	stParDutyCycle.fMinimum 		:= 0 		;
	stParDutyCycle.fMaximum			:= 50 		;
	stParDutyCycle.nNumber 			:= nLocationId + 2;
	stParDutyCycle.sDiscription  	:= CONCAT( STR1 := sName, STR2 := 'Percentage of period length in which an output is active');
	stParDutyCycle.sName			:= CONCAT( STR1 := sName, STR2 := 'Duty Cyle');
	stParDutyCycle.sType			:= 'MPar';
	stParDutyCycle.sUnit			:= '%';
	stParPeriodLength.fValue		:= 10;

	
	stParSwitchOverTime.fMinimum 	:= 0 		;
	stParSwitchOverTime.fMaximum	:= 500 		;
	stParSwitchOverTime.nNumber 	:= nLocationId + 3;
	stParSwitchOverTime.sDiscription:= CONCAT( STR1 := sName, STR2 := 'Idle time between output chanel switchover in miliseconds');
	stParSwitchOverTime.sName		:= CONCAT( STR1 := sName, STR2 := 'Switch Time');
	stParSwitchOverTime.sType		:= 'CPar';
	stParSwitchOverTime.sUnit		:= 'ms';

	stMaxTimeOn.fMinimum 	:= 0 		;
	stMaxTimeOn.fMaximum	:= 5000 	;
	stMaxTimeOn.nNumber 	:= nLocationId + 4;
	stMaxTimeOn.sDiscription:= CONCAT( STR1 := sName, STR2 := 'Maximum time a heater can be fully on without burning through');
	stMaxTimeOn.sName		:= CONCAT( STR1 := sName, STR2 := 'Max heating time');
	stMaxTimeOn.sType		:= 'MPar';
	stMaxTimeOn.sUnit		:= 'ms';
	
	
	// add parameters to handler 
	refFbParHandler.CmdAddParameter( refParameter := stParPeriodLength );
	refFbParHandler.CmdAddParameter( refParameter := stParDutyCycle );
	refFbParHandler.CmdAddParameter( refParameter := stParSwitchOverTime );
	
// ====== Set init status bit =======
	bInitOk := TRUE ;
END_METHOD

END_FUNCTION_BLOCK

// ---- Encoders/FunctionBlocks/FB_EncoderBase.TcPOU
{attribute 'reflection'}
FUNCTION_BLOCK PUBLIC FB_EncoderBase EXTENDS FB_DevBase
VAR_INPUT
END_VAR
VAR_OUTPUT
	{attribute 'analysis' := '-33'}
	nOutPosition		: LREAL	:= 0	; // Scaled position output
	{attribute 'analysis' := '-33'}
	nOutRaw				: UDINT := 0	; // Raw output value
	{attribute 'analysis' := '-33'}
	nVelocity			: LREAL	:= 0 	; // Velocity [units/sec]
END_VAR
VAR
	fPulsesPerUnit		: LREAL := 1	; // Scale factor for output [units/pulse]
	fOffset				: LREAL := 0	; // Offset for output
	bIcfInverted		: BOOL	:= FALSE; // Invert output position = standard false  
END_VAR

METHOD PUBLIC FastTask : BOOL
VAR_INPUT
END_VAR
END_METHOD

METHOD PUBLIC Init : BOOL
VAR_INPUT
	// Message location data
	nId			: UDINT ; // Identification number of object
	nParentId	: UDINT ; // Id of higher level If aplicable (0 = no parent)
	// Configuration
	fPulsesPerUnit	: LREAL	; // Scale factor for output [units/pulse]
	fOffset			: LREAL	; // Offset for output
	bIcfInverted	: BOOL	; // Invert output position = standard false  
END_VAR


// ====== Calculate device id =====
	ExecIdentifyDevice(nId,nParentId, E_ComponentTypes.Encoder);

// ====== Set manual device type ======
	eDevType := E_Devices.Encoder ;	

	
// ===== Coppy values to function memory ======
	THIS^.fPulsesPerUnit	:= MAX(fPulsesPerUnit,0.01); // Minimum value of 1
	THIS^.fOffset			:= fOffset;
	THIS^.bIcfInverted		:= bIcfInverted;
	
	
bInitOk := TRUE ;
END_METHOD

END_FUNCTION_BLOCK

// ---- Axis/FunctionBlocks/Analog/FB_DevAnalogAxis.TcPOU
FUNCTION_BLOCK PUBLIC FB_DevAnalogAxis EXTENDS FB_DevBase
VAR_INPUT
	stManualCtrl 	: ST_ManualAnalogAxisCtrl ; // Manual control
END_VAR
VAR_OUTPUT
	bDriveOk		: BOOL ; // Drive is ok
	bMovingCW		: BOOL ; // Move CW output is active
	bMovingCCW		: BOOL ; // Move CCW output is active
	fActVelocity	: LREAL; // Command velocity of motor
END_VAR
VAR // internal functions 
	fbVelocity		: FB_DevAnalogOutputScaled 	;
	fbqRun			: FB_DevDigitalOutput		;
	fbqReset		: FB_DevDigitalOutput		;
	fbqReverse		: FB_DevDigitalOutput		;
	fbiEnabled		: Fb_DevDigitalInput		;
END_VAR
VAR // Internal commands
	fCmdVelocity	: LREAL;
	bCmdRunCW 		: BOOL ;
	bCmdRunCCW		: BOOL ;
	bCmdReset		: BOOL ;	 
	bInternalEnable : BOOL ;
END_VAR

SUPER^(refFbFault := refFbFault);

// ===== Check inputs =====
	fbiEnabled( bEmbeded	:= TRUE,
				refFbFault 	:= refFbFault);

IF bInitOk THEN 
	ExecSetOutputs() ;
	bDriveOk	:= fbiEnabled.bFcoInputActive ;
END_IF

METHOD PUBLIC CmdManual : BOOL
VAR_INPUT
END_VAR
bCmdManual := TRUE ;

// Execute Manual commands
	IF stManualCtrl.bCmdRunCW THEN 
		CmdRunCW(fCmdVelocity := stManualCtrl.fCmdVelocity);
	ELSIF stManualCtrl.bCmdRunCCW THEN 
		CmdRunCCW(fCmdVelocity := stManualCtrl.fCmdVelocity);
	END_IF
END_METHOD

METHOD PUBLIC CmdReset : BOOL
VAR_INPUT
END_VAR
bErrorActive 	:= FALSE;

bCmdReset		:= TRUE ;

CmdReset		:= TRUE ;
END_METHOD

METHOD PUBLIC CmdRunCCW : BOOL
VAR_INPUT
	fCmdVelocity	: LREAL ; // Command velocity
END_VAR
bCmdRunCCW			:= TRUE ;
THIS^.fCmdVelocity 	:= fCmdVelocity ; 

CmdRunCCW 	:= bMovingCW ;
END_METHOD

METHOD PUBLIC CmdRunCW : BOOL
VAR_INPUT
	fCmdVelocity	: LREAL ; // Command velocity
END_VAR
bCmdRunCW := TRUE ;
THIS^.fCmdVelocity 	:= fCmdVelocity ;

CmdRunCW 	:= bMovingCW ;
END_METHOD

METHOD PUBLIC CmdSafeStop : BOOL
VAR_INPUT
END_VAR
bIsSafe := TRUE ;

bIsSafe := fbVelocity.CmdSafeStop() AND bIsSafe ;
bIsSafe := fbqRun.CmdSafeStop() 	AND bIsSafe ;
bIsSafe := fbqReverse.CmdSafeStop() AND bIsSafe ;
bIsSafe := fbqReset.CmdSafeStop() 	AND bIsSafe ;

CmdSafeStop := bIsSafe;
END_METHOD

METHOD PRIVATE ExecSetOutputs : BOOL
VAR_INPUT
END_VAR
// ====== Check safety and enable ======
IF bSafetyOk 
AND fbiEnabled.bFcoInputActive 
AND (bEnable OR bManual) THEN 
	bInternalEnable := TRUE;
ELSE
	fCmdVelocity 	:= 0;
	bCmdRunCW		:= FALSE;
	bCmdRunCCW		:= FALSE;
END_IF 

// ====== Set outputs =======
	fbVelocity	(	bEmbeded 	:= TRUE,
					bSafetyOk	:= bSafetyOk,
					bEnable		:= bInternalEnable,
					fCmdValue	:= fCmdVelocity, 
					refFbFault	:= refFbFault);
				
	fbqRun		(	bEmbeded 	:= TRUE,
					bSafetyOk	:= bSafetyOk,
					bEnable		:= bInternalEnable,
					bCmdOn		:= bCmdRunCW OR bCmdRunCCW,
					refFbFault	:= refFbFault);
				
	fbqReverse	(	bEmbeded 	:= TRUE,
					bSafetyOk	:= bSafetyOk,
					bEnable		:= bInternalEnable,
					bCmdOn		:= bCmdRunCCW,
					refFbFault	:= refFbFault);

	fbqReset	(	bEmbeded 	:= TRUE,
					bSafetyOk	:= bSafetyOk,
					bEnable		:= bInternalEnable,
					bCmdOn		:= bCmdReset,
					refFbFault	:= refFbFault);

// ===== reset input commands =====
	fCmdVelocity 	:= 0;
	bCmdRunCW		:= FALSE;
	bCmdRunCCW		:= FALSE;
	bCmdManual		:= FALSE;
	bCmdReset		:= FALSE;
	bInternalEnable := FALSE;
// ===== set feedback =====

bMovingCW		:= fbqRun.bOutputState AND NOT fbqReverse.bOutputState;
bMovingCCW		:= fbqRun.bOutputState AND fbqReverse.bOutputState;
fActVelocity	:= fbVelocity.fOutputValue ;
END_METHOD

METHOD Init : BOOL
VAR_INPUT
	// Message location data
	nId			: UDINT ; // Identification number of object
	nParentId	: UDINT ; // Id of higher level If aplicable (0 = no parent)

	// Motor settings
	fMaxVelocity : LREAL ; // Maximum motor velocity for scaling
END_VAR
// ====== initialize components =====
	bInitOk := TRUE ;

// ====== Calculate device id =====
	bInitOk :=	ExecIdentifyDevice(nId,nParentId, E_ComponentTypes.Axis) AND bInitOk;

// ====== Set manual device type ======
	eDevType := E_Devices.AnalogAxis ;	


bInitOk := 	fbVelocity.Init	( 	nId 			:= 0,
								nParentId		:= nLocationId,
								benableNegative	:= FALSE )
								AND bInitOk;
			fbVelocity.SetScaling	(fMaxValue 		:= fMaxVelocity);
								
bInitOk	:= 	fbqRun.Init		( 	nId				:= 1,
								nParentId		:= nLocationId)
								AND bInitOk;

bInitOk	:= 	fbqReset.Init	( 	nId				:= 2,
								nParentId		:= nLocationId)
								AND bInitOk;

bInitOk	:= 	fbqReverse.Init	( 	nId				:= 3,
								nParentId		:= nLocationId)
								AND bInitOk;

bInitOk	:= 	fbiEnabled.Init	( 	nId				:= 4,
								nParentId		:= nLocationId)
								AND bInitOk;

// ====== Set feedback =======
Init := bInitOk;
END_METHOD

END_FUNCTION_BLOCK

// ---- Outputs/AnalogOutputs/FB_DevAnalogOutputScaled.TcPOU
{attribute 'reflection'}
FUNCTION_BLOCK FB_DevAnalogOutputScaled EXTENDS FB_DevAnalogOutput
VAR_INPUT
END_VAR
VAR_OUTPUT
END_VAR
VAR
	fGainFactor 	: LREAL:= 32767	;
END_VAR

SUPER^(refFbFault := refFbFault);

METHOD INTERNAL ExecSetFeedback : BOOL
VAR_INPUT
END_VAR
// Set feedback 
fOutputValue := qnHwOut ;
END_METHOD

METHOD INTERNAL ExecSetOutput : BOOL
VAR_INPUT
END_VAR
// Set Output to physical device
IF bSafetyOk AND (bEnable OR bCmdManual) THEN 
	qnHwOut := LREAL_TO_INT(fCmdValue * fGainFactor) ;
	qnHwOut := LIMIT(nLimitMin, qnHwOut, nLimitMax) ; 
ELSE 
	qnHwOut		:= 0;
	fCmdValue 	:= 0 ; 
END_IF
END_METHOD

METHOD PUBLIC SetScaling : BOOL 
VAR_INPUT
	fMaxValue	: LREAL ; 		// Maximum input value after scaling, e.g. 100% (mandatory input)  
END_VAR
// calculate gain 
fGainFactor := nLimitMax / fMaxValue ;
END_METHOD

END_FUNCTION_BLOCK

// ---- Axis/FunctionBlocks/ServoHybrid/FB_DevBasicACAxis.TcPOU
{attribute 'reflection'}
FUNCTION_BLOCK PUBLIC FB_DevBasicACAxis EXTENDS FB_DevBase
VAR_INPUT
	// ===== General Function input =====
		fCmdAcc			: LREAL := 15000;
		fCmdDecc		: LREAL := 15000; 
	// Manual control reference
		stManualCtrl	: UDT_ManualAxisCtrl ;
END_VAR
VAR_OUTPUT
	bHomed			: BOOL 	:= FALSE; 
	bMoving		: BOOL ; // Axis is moving
	bInPosition : BOOL ; // Axis is in position 
END_VAR
VAR
		AxisRef	: AXIS_REF ; // reference to AC axis
	// ===== HW Config Bits =====
		bIcfCmdVelocityRpm	: BOOL ; // input speeds in Rpm
		bIcfEnableForward 	: BOOL ; // Enable forward motion
 		bIcfEnablereverse	: BOOL ; // Enable reverse motion
		bIcfAlwaysEnable	: BOOL ; // 1 = Axis always enabled, 0 = Axis disabled at Idle 
		bIcfSimulationMode	: BOOL := FALSE ; // Simulation mode is active [default set to False] 
	// ===== Internal motion values ======
		fHomePosition		: LREAL := 0 ; // set position at homing
	// ====== Axis Settings ======
		fMaxVelo		: LREAL := 0 ; // Axis Maximum velocity
		fMaxAcc			: LREAL := 0 ; // Axis Maximum cceleration
		fMaxDec			: LREAL := 0 ; // axis Maxium deceleration 
		
		fSafeVeloLimit	: LREAL	:= 200; // Safe velocity limit 
		tEnableDelay	: TIME 	:= T#150MS	;
		tDisableDelay	: TIME 	:= T#500MS  ;
		
	// ====== Axis enable =====	
		bCmdEnableAxis 		: BOOL 	:= FALSE; // Command to enable the axis (External)
		bInternalEnable		: BOOL 	:= FALSE; // internal enable command (turns off after set time, and on at new motion command
		bDelayedEnable		: BOOL 	:= false; // Delayed enable signal for motion commands
		TonMotionEnable		: TON 			; // Timer on for motion command enable
		TofIntAxisEnable	: TOF  			; // Timer off for internal axis enable 
	// ===== Safe commands =====
		bCmdSafeStop	: BOOL ;
	// Motion commands 
		fbMcPower 			: MC_Power		;		// FB for enable and override
		fbMcReset 			: MC_Reset		;		// FB to reset axis
		fbSoeReset			: FB_SoEReset	; 		// FB to reset axis hardware
		fbMcHome			: MC_Home		;		// Fb to home Axis
		fbMcStop 			: MC_Stop		;		// FB to stop axis
		fbMcHalt			: MC_Halt		;		// FB to halt axis
		fbMcJog				: MC_Jog		;		// FB to Jog axis
		fbMcMoveVelocity	: MC_MoveVelocity;		// FB to move with specified velocity until Next command is given
	(* PtoP Motion move commands are in arrays so multiple commands can be stacked *) 
		fbMCMoveRelative	: ARRAY [0..1] OF MC_MoveRelative	;		// FB to move relative
		fbMcMoveAbsolute	: ARRAY [0..1] OF MC_MoveAbsolute	;		// FB to move axis (velocity movement)
		
	// Parameters 
		stMParMaxAcc : Udt_Parameter := (fMaximum := 999999, fMinimum := 0, fValue := 0)	; // Parameter for maximum acceleration
		stMParMaxDec : Udt_Parameter := (fMaximum := 999999, fMinimum := 0, fValue := 0)	; // Parameter for maximum Deceleration
		stMparMaxVelo: Udt_Parameter := (fMaximum := 999999, fMinimum := 0, fValue := 0)	; // Parameter for maximum velocity
		
	// Device feedback
		nActVelocity AT%I* : INT ; // actual speed of the motor
		nActPosition AT%I* : UDINT ; // Actual position of the motor

	// ===== Function execute triggers =====
		bExec_Reset			: BOOL := FALSE; // Execute reset
		bExec_Halt			: BOOL := FALSE; // Execute hold
		bExec_Home			: BOOL := FALSE; // Execute Home
		bExec_JogPositive	: BOOL := FALSE; // Execute Jog in positive direction
		bExec_JogNegative	: BOOL := FALSE; // Execute Jog in negative direction
		bExec_MoveVelocity	: BOOL := FALSE; // Execute move velocity
		arExec_MoveRelative	: ARRAY [0..1] OF BOOL ; // Execute move relative
		arExec_MoveAbs		: ARRAY [0..1] OF BOOL ; // Execute move absolute reverse
		

END_VAR

// Call base function
SUPER^(refFbFault := refFbFault);

// ==== Check if axis is initiated =====
IF NOT bInitOk THEN 
	RETURN ; 
END_IF

// ===== Execute safe functions =====
	ExecSafeFunctions(); 

// ==== Execute organizational functions =====
	ExecEnable();

// ==== execute motion functions =====
	CallMotionFunctions();

METHOD PRIVATE CallMotionFunctions : BOOL
VAR_INPUT
END_VAR
// ===== Check if safe to move =====
	IF bCmdSafeStop OR NOT bDelayedEnable THEN 
		RETURN ;
	END_IF

// ===== Homing functions =====
	ExecHome		(); 

// ===== Motion standstil commands =====
	ExecHalt		();

// ===== Motion move functions
	ExecJog			(); 
	ExecMoveAbsolute();
	ExecMoveRelative();
	ExecMoveVelocity();
END_METHOD

METHOD PUBLIC CmdHalt : BOOL
VAR_INPUT
	fDeceleration 	: LREAL := 0 ; // command deceleration
	mcBuffermode	: MC_BufferMode ; // Buffermode defines how the previous command is executed.
END_VAR
// Set command to true 
bExec_Halt 		:= TRUE ;
bInternalEnable	:= TRUE ;

// coppy parameters
fbMcHalt.Deceleration	:= fDeceleration;
fbMcHalt.BufferMode		:= mcBuffermode	;

// Set feedback output 
CmdHalt := fbMchalt.Active ;
END_METHOD

METHOD PUBLIC CmdHome : BOOL // start axis homing procedure
VAR_INPUT
	fPosition 		: LREAL := 0 ; // Homing position
	mcBufferMode	: MC_BufferMode := MC_BufferMode.MC_Aborting		; // Buffermode
END_VAR
// set command to true 
bExec_Home 		:= TRUE	; 
bInternalEnable	:= TRUE ;

// coppy parameters
fbMcHome.Position 	:= fPosition 	;
fbMcHome.BufferMode	:= mcBufferMode ;

// Set feedback output
CmdHome := fbMcHome.Done ;
END_METHOD

METHOD PUBLIC CmdJog : BOOL // Jog axis with variable speed. jog stops as soon as the command is false
VAR_INPUT
	fVelocity		: LREAL 	; // jog velocity can be adjusted as long as the command is active
	fPos			: LREAL 	; // Jog position or step size (if aplicable)
	bJogNegative 	: BOOL 		:= FALSE ; // jog in negative direction
	eJogmode		: E_JogMode := E_JogMode.MC_JOGMODE_CONTINOUS ; // jogmode [default MC_JOGMODE_CONTINOUS] 
END_VAR
// Velocity conversion from RPM to deg/sec
	IF bIcfCmdVelocityRpm THEN 
		fVelocity := Rpm_To_DegS(fVelocity);
	END_IF

// Set command to true
	IF fbMcJog.Velocity = fVelocity THEN // If command velocity changes, then set exec to false for one cycle to trigger new velocity so the jog follows the set velocity
		bExec_JogPositive	:= NOT bJogNegative ;
		bExec_JogNegative 	:= bJogNegative ;
	END_IF
	bInternalEnable			:= TRUE ;

// coppy parameters
	fbMcJog.Velocity	:= fVelocity 	;
	fbmcjog.Mode		:= eJogmode		;
	fbMcJog.Position	:= fPos			;

// Set feedback output 
	CmdJog := fbMcJog.Active ;
END_METHOD

METHOD PUBLIC CmdManual : BOOL
VAR
	eJogmode		: E_JogMode := E_JogMode.MC_JOGMODE_CONTINOUS ; // jogging mode 
END_VAR
// Enable axis for manual control
bCmdManual := TRUE ;

// set jog mode 
IF stManualCtrl.bCmdInching THEN 
	eJogmode := E_JogMode.MC_JOGMODE_INCHING ;
END_IF

// execute motion commands
IF stManualCtrl.bCmdJogForward OR stManualCtrl.bCmdJogReverse THEN 
	CmdJog (fVelocity := stManualCtrl.fVelocity, 
			fPos := stManualCtrl.fDistance, 
			bJogNegative := stManualCtrl.bCmdJogReverse, 
			eJogmode := eJogmode);
ELSIF stManualCtrl.bCmdToPos THEN 
	CmdMoveAbs( fPosition := stManualCtrl.fPosition, 
				fVelocity := stManualCtrl.fVelocity, 
				mcBuffermode := MC_BufferMode.MC_Aborting);
ELSIF stManualCtrl.bCmdHome THEN 
	CmdHome( fPosition := 0, mcBufferMode := MC_Aborting);
ELSE 
	CmdHalt( 	fDeceleration := fMaxDec * 0.9, 
				mcBuffermode := MC_BufferMode.MC_Aborting) ; 
END_IF
END_METHOD

METHOD PUBLIC CmdMoveAbs : BOOL // Move absolute command
VAR_INPUT
	fPosition	:	LREAL 	; // target position
	fVelocity	: 	LREAL 	; // Maximum velocity [units/sec]
	mcBuffermode: 	MC_BufferMode ; // Buffermode defines how the previous command is executed.
END_VAR
// Velocity conversion from RPM to deg/sec
	IF bIcfCmdVelocityRpm THEN 
		fVelocity := Rpm_To_DegS(fVelocity);
	END_IF

// Determine function for command stacking
	IF fbMcMoveAbsolute[0].Active THEN 
		arExec_MoveAbs[1] 				:= (fPosition <> fbMcMoveAbsolute[0].Position OR fVelocity <> fbMcMoveAbsolute[0].Velocity) ;
		fbMcMoveAbsolute[1].Position 	:= fPosition ;
		fbMcMoveAbsolute[1].Velocity 	:= fVelocity ; 
		fbMcMoveAbsolute[1].BufferMode 	:= mcBuffermode ;
	ELSE
		arExec_MoveAbs[0] 				:= (fPosition <> fbMcMoveAbsolute[1].Position OR fVelocity <> fbMcMoveAbsolute[1].Velocity) ;
		fbMcMoveAbsolute[0].Position 	:= fPosition ;
		fbMcMoveAbsolute[0].Velocity 	:= fVelocity ; 
		fbMcMoveAbsolute[0].BufferMode 	:= mcBuffermode ;
	END_IF

bInternalEnable	:= TRUE ;
// set feedback
IF arExec_MoveAbs[1] OR fbMcMoveAbsolute[1].Busy THEN 
	CmdMoveAbs :=	fbMcMoveAbsolute[1].Active ;
ELSE 
	CmdMoveAbs :=	fbMcMoveAbsolute[0].Active ;
END_IF
END_METHOD

METHOD CmdMoveRelative : BOOL // move relative command 
VAR_INPUT
	fDistance	:	LREAL 	; // target position
	fVelocity	: 	LREAL 	; // Maximum velocity [units/sec]
	mcBuffermode: 	MC_BufferMode ; // Buffermode defines how the previous command is executed.
END_VAR
// Velocity conversion from RPM to deg/sec
	IF bIcfCmdVelocityRpm THEN 
		fVelocity := Rpm_To_DegS(fVelocity);
	END_IF

// Determine function for command stacking
	IF fbMCMoveRelative[0].Active THEN 
		arExec_MoveRelative[1] := (fDistance <> fbMCMoveRelative[0].Distance OR fVelocity <> fbMCMoveRelative[0].Velocity) ;
		fbMCMoveRelative[1].Velocity	:= fVelocity 	;
		fbMCMoveRelative[1].Distance	:= fDistance	;
		fbMCMoveRelative[1].BufferMode	:= mcBuffermode	;
	ELSE 
		arExec_MoveRelative[0] := (fDistance <> fbMCMoveRelative[1].Distance OR fVelocity <> fbMCMoveRelative[1].Velocity) ;
		fbMCMoveRelative[0].Velocity	:= fVelocity 	;
		fbMCMoveRelative[0].Distance	:= fDistance	;
		fbMCMoveRelative[0].BufferMode	:= mcBuffermode	;
	END_IF

bInternalEnable	:= TRUE ;

// set feedback
IF arExec_MoveRelative[1] OR fbMCMoveRelative[1].Busy THEN 
	CmdMoveRelative :=	fbMCMoveRelative[1].Active ;
ELSE
	CmdMoveRelative :=	fbMCMoveRelative[0].Active ;
END_IF
END_METHOD

METHOD PUBLIC CmdMoveVelocity : BOOL // Move with set velocity until stopped
VAR_INPUT
	fVelocity	: 	LREAL 	; // Maximum velocity [units/sec]
	mcDirection : 	MC_Direction := MC_Direction.MC_Positive_Direction ; // Direction of movement mc_direction [ deafult mc_positive_direction]
	mcBuffermode: 	MC_BufferMode ; // Buffermode defines how the previous command is executed.
END_VAR
// Velocity conversion from RPM to deg/sec
	IF bIcfCmdVelocityRpm THEN 
		fVelocity := Rpm_To_DegS(fVelocity);
	END_IF

// Set command to true 
	bExec_MoveVelocity 	:= TRUE ;
	bInternalEnable		:= TRUE ;

// coppy parameters
	fbMcMoveVelocity.Velocity	:= fVelocity 	;
	fbMcMoveVelocity.Direction 	:= mcDirection	;
	fbMcMoveVelocity.BufferMode	:= mcBuffermode	;

// Set feedback output 
	CmdMoveVelocity := fbMcMoveVelocity.Active ;
END_METHOD

METHOD PUBLIC CmdReset : BOOL
VAR_INPUT
END_VAR
// Set reset axis to true 				
	bExec_Reset 	:= TRUE ; 
	bInternalEnable	:= TRUE ;
	
// Set feedback output 
	CmdReset := fbMcReset.Done ;
END_METHOD

METHOD PUBLIC CmdSafeStop : BOOL
VAR_INPUT
END_VAR
// Set safestop command
bCmdSafeStop := TRUE ; 

// Set feedback output 
CmdSafeStop := bIsSafe OR NOT bInitOk;
END_METHOD

METHOD PRIVATE ExecEnable : BOOL
VAR_INPUT
END_VAR
// ===== Set axis enable ======
IF NOT bEnable AND NOT bCmdManual AND nActVelocity <> 0 THEN
	CmdHalt(fDeceleration := fCmdDecc, mcBuffermode := MC_BufferMode.MC_Aborting);
ELSE 
	bCmdEnableAxis	:= bEnable OR bCmdManual ;
	bCmdManual := FALSE ;
END_IF

// ===== Check if axis is bussy with a command =====
	bInternalEnable	S= bIcfAlwaysEnable ; // always enable axis if configured
	
// ===== Axis disable timer after last command =====
	TofIntAxisEnable (	IN:= bInternalEnable, PT := tDisableDelay);

// ===== Enable drive =====
	fbMcPower(	Axis			:= AxisRef , 
				Enable			:= bCmdEnableAxis AND TofIntAxisEnable.Q, 
				Enable_Positive	:= bIcfEnableForward, 
				Enable_Negative	:= bIcfEnablereverse, 
				Override		:= 100 );  
				
// ===== Reset internal enable signal =====
	bInternalEnable := FALSE ; 	

// ===== Delayed enable function =====	
	TonMotionEnable(IN := fbMcPower.Active, PT := tEnableDelay);
	bDelayedEnable := TonMotionEnable.Q ;	


IF fbMcPower.Error THEN 
	bErrorActive			:= TRUE							;
	stFault.Active 			:= TRUE 						;
	stFault.MessageNumber	:= E_MessageNumbers.FF_AxisFault;
	stFault.Discription		:= CONCAT('Enable Fault ', UDINT_TO_STRING(fbMcPower.ErrorID));				;
	stFault.FaultType		:= E_FaultTypes.FF				;
END_IF
END_METHOD

METHOD PRIVATE ExecHalt : BOOL
VAR_INPUT
END_VAR
// ==== Execute halt function ===== 
fbMcHalt (	Axis 		:= AxisRef,
			Execute 	:= bExec_Halt );

// ===== reset command =====
	bExec_Halt := FALSE ;
	bInternalEnable := fbMcHalt.Busy ;			
	
// Halt fault handling 
	IF fbMcHalt.Error THEN 
		bErrorActive			:= TRUE							;
		stFault.Active 			:= TRUE 						;
		stFault.MessageNumber	:= E_MessageNumbers.FF_AxisFault;
		stFault.Discription		:= CONCAT('Halt Fault ', UDINT_TO_STRING(fbMcHalt.ErrorID));				;
		stFault.FaultType		:= E_FaultTypes.FF				;
	END_IF
END_METHOD

METHOD PRIVATE ExecHome : BOOL
VAR_INPUT
END_VAR
// ==== execute homing function =====
	fbMcHome(	Axis			:= AxisRef,
				Execute			:= bExec_Home,
				HomingMode		:= MC_DefaultHoming ); 
			
// Reset exec command 
	bExec_Home 	:= FALSE ;
	bHomed		S= fbMcHome.Done ;	
	bInternalEnable := fbMcHome.Busy ;			
				
// fault handling 
	IF fbMcHome.Error THEN 
		bErrorActive			:= TRUE							;
		stFault.Active 			:= TRUE 						;
		stFault.MessageNumber	:= E_MessageNumbers.FF_AxisFault;
		stFault.Discription		:= CONCAT('Homing Fault ', UDINT_TO_STRING(fbMcHome.ErrorID));				;
		stFault.FaultType		:= E_FaultTypes.FF				;
	END_IF
END_METHOD

METHOD PRIVATE ExecJog : BOOL
VAR_INPUT
END_VAR
// ===== Execute Jog function =====
	// function call
	fbMcJog (	Axis 		:= AxisRef,
				JogForward	:= bExec_JogPositive,
				JogBackwards:= bExec_JogNegative,
				Acceleration:= fCmdAcc,
				Deceleration:= fCmdDecc );

// ===== reset command =====
	bExec_JogPositive 	:= FALSE  ;
	bExec_JogNegative	:= FALSE  ;
	bInternalEnable		:= fbMcJog.Busy; 

// Jog fault handling 
	IF fbMcJog.Error THEN 
		bErrorActive			:= TRUE							;
		stFault.Active 			:= TRUE 						;
		stFault.MessageNumber	:= E_MessageNumbers.FF_AxisFault;
		stFault.Discription		:= CONCAT('Jog Fault ', UDINT_TO_STRING(fbMcJog.ErrorID));				;
		stFault.FaultType		:= E_FaultTypes.FF				;
	END_IF
END_METHOD

METHOD PRIVATE ExecMoveAbsolute : BOOL
VAR_INPUT
END_VAR
VAR
	i : UDINT := 0 ;
END_VAR
// ==== execute move absolute function =====
FOR i := 0 TO 1 DO 
	// function call
	fbMcMoveAbsolute[i](	Axis 		:= AxisRef,
							Execute 	:= arExec_MoveAbs[i],
							Acceleration:= fCmdAcc,
							Deceleration:= fCmdDecc );  
	// reset Exec command 
	arExec_MoveAbs[i] := FALSE ; 
	bInternalEnable := fbMcMoveAbsolute[i].Busy ;			

	// If function is done then reset command values
	IF fbMcMoveAbsolute[i].Done THEN 
		fbMcMoveAbsolute[i].Velocity	:= 0 ;
		fbMcMoveAbsolute[i].Position	:= 0 ; 
	END_IF
	
	// fault handling 
	IF fbMcMoveAbsolute[i].Error THEN 
		bErrorActive			:= TRUE							;
		stFault.Active 			:= TRUE 						;
		stFault.MessageNumber	:= E_MessageNumbers.FF_AxisFault;
		stFault.Discription		:= CONCAT('Move absolute Fault ', UDINT_TO_STRING(fbMcMoveAbsolute[i].ErrorID));				;
		stFault.FaultType		:= E_FaultTypes.FF				;
	END_IF
END_FOR
END_METHOD

METHOD PRIVATE ExecMoveRelative : BOOL
VAR_INPUT
END_VAR
VAR
	i : UDINT := 0 ;
END_VAR
// ===== Execute move relative function ======
FOR i := 0 TO 1 DO 
	// function call
	fbMCMoveRelative[i](	Axis 		:= AxisRef,
							Execute		:= arExec_MoveRelative[i],
							Acceleration:= fCmdAcc,
							Deceleration:= fCmdDecc );
	// reset Exec command 
	arExec_MoveRelative[i] := FALSE ; 
	bInternalEnable := fbMCMoveRelative[i].Busy ;			

	// If function is done then reset command values
	IF fbMCMoveRelative[i].Done THEN 
		fbMCMoveRelative[i].Velocity	:= 0 ;
		fbMCMoveRelative[i].Distance	:= 0 ; 
	END_IF
	
	// fault handling 
	IF fbMCMoveRelative[i].Error THEN 
		bErrorActive			:= TRUE							;
		stFault.Active 			:= TRUE 						;
		stFault.MessageNumber	:= E_MessageNumbers.FF_AxisFault;
		stFault.Discription		:= CONCAT('Move relative Fault ', UDINT_TO_STRING(fbMCMoveRelative[i].ErrorID));				;
		stFault.FaultType		:= E_FaultTypes.FF			;
	END_IF
END_FOR
END_METHOD

METHOD PRIVATE ExecMoveVelocity : BOOL
VAR_INPUT
END_VAR
// ===== Execute move velocity function =====
// function call
fbMcMoveVelocity (	Axis 		:= AxisRef,
					Execute		:= bExec_MoveVelocity,
					Acceleration:= fCmdAcc,
					Deceleration:= fCmdDecc );

// ===== reset command =====
bExec_MoveVelocity := FALSE ;
bInternalEnable		:= fbMcMoveVelocity.Busy;
	
// Halt fault handling 
IF fbMcHalt.Error THEN 
	bErrorActive			:= TRUE							;
	stFault.Active 			:= TRUE 						;
	stFault.MessageNumber	:= E_MessageNumbers.FF_AxisFault;
	stFault.Discription		:= CONCAT('Move velocity Fault ', UDINT_TO_STRING(fbMcMoveVelocity.ErrorID));				;
	stFault.FaultType		:= E_FaultTypes.FF				;
END_IF
END_METHOD

METHOD PRIVATE ExecReset : BOOL
VAR_INPUT
END_VAR
IF  nActVelocity <> 0 AND bExec_Reset THEN // If the axis is still moving execute safe stop first
	CmdSafeStop();
	RETURN;
END_IF

// perform reset 
	fbMcReset	( 	Execute	:= bexec_reset AND NOT fbSoeReset.Busy,
					Axis	:= AxisRef ); 
					
// ===== reset command =====
	bExec_Reset := FALSE ;
	
// ===== reset internal fault bits and stop bits =====
	bErrorActive 			:= FALSE ; 
	
// ===== reset safe commands ======
	bCmdSafeStop	:= FALSE ; 
	
// Reset fault handling 
	IF fbSoeReset.Error OR fbMcReset.Error THEN 
		bErrorActive			:= TRUE							;
		stFault.Active 			:= TRUE 						;
		stFault.MessageNumber	:= E_MessageNumbers.FF_AxisFault;
		stFault.Discription		:= CONCAT('Reset Fault ', UDINT_TO_STRING(fbMcReset.ErrorID))			;
		stFault.FaultType		:= E_FaultTypes.FF				;
	END_IF
END_METHOD

METHOD PRIVATE ExecSafeFunctions : BOOL
VAR_INPUT
END_VAR
// ==== Stop when safety is not ok =====
	bCmdSafeStop := NOT bSafetyOk ;

// ==== Safe operation functions (overrule all other motion functions) =====
	fbMcStop( 	Axis 			:= AxisRef		,
				Execute 		:= bCmdSafeStop	,
				Deceleration	:= fMaxDec		);
	
	// Reset axis command			
	bCmdSafeStop 	R= fbMcStop.Done ;
	
// Safestop fault handling 
	IF fbMcStop.Error THEN 
		bErrorActive			:= TRUE							;
		stFault.Active 			:= TRUE 						;
		stFault.MessageNumber	:= E_MessageNumbers.FF_AxisFault;
		stFault.Discription		:= CONCAT('Safe stop axis fault ', UDINT_TO_STRING(fbMcStop.ErrorID));				;
		stFault.FaultType		:= E_FaultTypes.FF				;
	END_IF

// ===== Dev is safe feedback =====
bIsSafe := NOT bCmdEnableAxis  ;
END_METHOD

METHOD PUBLIC Init : BOOL
VAR_INPUT
	// Message location data
	nId			: UDINT ; // Identification number of object
	nParentId	: UDINT ; // Id of higher level If aplicable (0 = no parent)
	// Config Bits
	bIcfCmdVelocityRpm	: BOOL := FALSE ; // input speeds in Rpm
	bIcfEnableForward 	: BOOL := TRUE 	; // Enable forward motion
	bIcfEnablereverse	: BOOL := TRUE 	; // Enable reverse motion
	bIcfAlwaysEnable	: BOOL := FALSE ; // 1 = Axis always enabled, 0 = Axis disabled at Idle 
	bIcfSimulationMode	: BOOL := FALSE ; // Simulation mode is active [default set to False] Used for testing without hardware present 
	
	fHomePosition		: LREAL := 0 	; // set position at homing
	fSafeVeloLimit		: LREAL	:= 360 	; // safe velocity limit [deg/sec]
	nEncTurnoverVal 	: LREAL := 360	; // encoder turnover value 
	tEnableDelay		: time 	:= T#0MS; // Time between axis enable command and motion command execution (0 := no delay active)	
	tDisabledelay		: TIME 	:= T#100MS; // Axis idle time before axis is disabled 
END_VAR
VAR 
	bActParamValid 		: BOOL ; // Parameter read is valid 
END_VAR
// ====== Set init to true =====
	bInitOk	:= TRUE ; 

// ====== Calculate device id =====
	bInitOk :=	ExecIdentifyDevice(nId,nParentId, E_ComponentTypes.Axis) AND bInitOk;

// ===== Message data set =====
	stFault.ComponentType		:= E_ComponentTypes.Axis ;
	
// ===== Write parameters =====
	stMParMaxAcc.nNumber		:= nLocationId + 1;
	stMParMaxAcc.sDiscription 	:= CONCAT(STR1 := sName, STR2:= ' hardware maximum accaleration (0 = HWMaximum)'); 
	stMParMaxAcc.sName			:= CONCAT(STR1 := sName, STR2:= 'Hard max aceleration');
	stMParMaxAcc.sType			:= 'MPar';
	stMParMaxAcc.sUnit			:= 'Units/Sec^2';
	
	stMParMaxDec.nNumber		:= nLocationId + 2;
	stMParMaxDec.sDiscription 	:= CONCAT(STR1 := sName, STR2:= ' hardware maximum deceleration(0 = HWMaximum)'); 
	stMParMaxDec.sName			:= CONCAT(STR1 := sName, STR2:= 'Hard max deceleration');
	stMParMaxDec.sType			:= 'MPar';
	stMParMaxDec.sUnit			:= 'Units/Sec^2';
	
	stMparMaxVelo.nNumber		:= nLocationId + 3;
	stMparMaxVelo.sDiscription 	:= CONCAT(STR1 := sName, STR2:= ' hardware maximum velocity'); 
	stMparMaxVelo.sName			:= CONCAT(STR1 := sName, STR2:= 'Hard max velocity');
	stMparMaxVelo.sType			:= 'MPar';
	stMparMaxVelo.sUnit			:= 'Units/Sec';

	refFbParHandler.CmdAddParameter(refParameter := stMParMaxAcc);
	refFbParHandler.CmdAddParameter(refParameter := stMParMaxDec);
	refFbParHandler.CmdAddParameter(refParameter := stMparMaxVelo);

// ===== set axis configuration =====	
	fMaxAcc	:= stMParMaxAcc.fValue;
	fMaxDec	:= stMParMaxDec.fValue;	
	fMaxVelo:= stMparMaxVelo.fValue;

	fCmdAcc 		:= fMaxAcc;
	fCmdDecc		:= fMaxDec;
// ===== Configure Axis =====
	// ***** Config Bits *****
		THIS^.bIcfCmdVelocityRpm	:= bIcfCmdVelocityRpm	; // Enable speed inputs in Rpm
		THIS^.bIcfEnableForward 	:= bIcfEnableForward 	; // Enable forward motion
		THIS^.bIcfEnablereverse		:= bIcfEnablereverse	; // Enable reverse motion
		THIS^.bIcfAlwaysEnable		:= bIcfAlwaysEnable		; // Always enable motor and brake if safety is ok
		THIS^.bIcfSimulationMode	:= bIcfSimulationMode 	; // Simulation mode is active [default set to False] 

	// ***** config homing Mode ***** 
 		THIS^.fHomePosition			:= fHomePosition;
	// ***** Velocity settings *****
		THIS^.fSafeVeloLimit 		:= fSafeVeloLimit ; // set maximum safe velocity	
	// ***** Time delay enable off *****
		THIS^.tEnableDelay		:= tEnableDelay	;
		THIS^.tDisableDelay 	:= tDisabledelay ;		

// ===== Set device type for manual control =====
	eDevType := E_Devices.Axis ;
		
// ===== reset axis state indicators ======
	bErrorActive 	:= FALSE;
END_METHOD

END_FUNCTION_BLOCK

// ---- Axis/FunctionBlocks/ServoHybrid/FB_DevHybridAc.TcPOU
{attribute 'reflection'}
FUNCTION_BLOCK PUBLIC FB_DevHybridAc EXTENDS Fb_DevAxis
VAR_INPUT
END_VAR
VAR_OUTPUT
END_VAR
VAR
	// Parameters 
		stMParMaxAcc : Udt_Parameter := (fMaximum := 999999, fMinimum := 0, fValue := 0)	; // Parameter for maximum acceleration
		stMParMaxDec : Udt_Parameter := (fMaximum := 999999, fMinimum := 0, fValue := 0)	; // Parameter for maximum Deceleration
		stMparMaxVelo: Udt_Parameter := (fMaximum := 999999, fMinimum := 0, fValue := 0)	; // Parameter for maximum velocity
END_VAR

SUPER^(refFbFault := refFbFault);

METHOD INTERNAL ExecHalt : BOOL
VAR_INPUT
END_VAR
// The hybrid axis is equiped with it's own safety stop system therefore mc halt is no longer needed with an Estop
IF bSafetyOk THEN 
	// ==== Execute halt function ===== 
	fbMcHalt (	Axis 		:= AxisRef,
				Execute 	:= bExec_Halt );
END_IF
// ===== reset command =====
	bExec_Halt := FALSE ;
	
// Halt fault handling 
	IF fbMcHalt.Error THEN 
		bError					:= TRUE							;
		stFault.Active 			:= TRUE 						;
		stFault.MessageNumber	:= E_MessageNumbers.FF_AxisFault;
		stFault.Discription		:= CONCAT('Halt Fault ', UDINT_TO_STRING(fbMcHalt.ErrorID));				;
		stFault.FaultType		:= E_FaultTypes.FF				;
	END_IF
END_METHOD

METHOD INTERNAL ExecReadStatus : BOOL
VAR_INPUT
END_VAR
// Read axis status from drive
AxisRef.ReadStatus();						
// convert velocity to RPM for output if aplicable
IF bIcfCmdVelocityRpm THEN 
	fVelocity := AxisRef.NcToPlc.ActVelo / 6 ;
ELSE 
	fVelocity := AxisRef.NcToPlc.ActVelo ;
END_IF

// write position output
fActPosition := AxisRef.NcToPlc.ActPos ;
						
// set status bits 
bIdle := NOT AxisRef.Status.HasJob ;
END_METHOD

METHOD INTERNAL ExecReset : BOOL
VAR_INPUT
END_VAR
IF  AxisRef.Status.Moving AND bExec_Reset THEN // If the axis is still moving execute safe stop first
	CmdSafeStop();
	RETURN;
END_IF

	fbMcReset	( 	Execute	:= bexec_reset,
					Axis	:= AxisRef ); 
					
// ===== reset command =====
	bExec_Reset := FALSE ;
	
// ===== reset internal fault bits and stop bits =====
	bError 			:= FALSE ; 
	
// ===== reset safe commands ======
	bCmdSafeStop	:= FALSE ; 
	bCmdSafeSpeed 	:= FALSE ;
	
// Reset fault handling 
	IF fbMcReset.Error THEN 
		bError					:= TRUE							;
		stFault.Active 			:= TRUE 						;
		stFault.MessageNumber	:= E_MessageNumbers.FF_AxisFault;
		stFault.Discription		:= CONCAT('Reset Fault ', UDINT_TO_STRING(fbMcReset.ErrorID))			;
		stFault.FaultType		:= E_FaultTypes.FF				;
	END_IF
END_METHOD

METHOD PUBLIC Init : BOOL
VAR_INPUT
	// Message location data
	nId			: UDINT ; // Identification number of object
	nParentId	: UDINT ; // Id of higher level If aplicable (0 = no parent)
	// Config Bits
	bIcfCmdVelocityRpm	: BOOL := FALSE ; // input speeds in Rpm
	bIcfEnableForward 	: BOOL := TRUE 	; // Enable forward motion
	bIcfEnablereverse	: BOOL := TRUE 	; // Enable reverse motion
	bIcfAlwaysEnable	: BOOL := FALSE ; // 1 = Axis always enabled, 0 = Axis disabled at Idle 
	bIcfSimulationMode	: BOOL := FALSE ; // Simulation mode is active [default set to False] Used for testing without hardware present 
	bIcfModuloAxis		: BOOL := FALSE ; // Show axis position as modulo
	bIcfSTOPresent		: BOOL := FALSE ; // Axis safe torque off is present	
	bIcfNCHomeSensor	: BOOL := FALSE ; // Homing sensor is inverted (NC)	

	// Config Values 
	mcHomingMode 		: MC_HomingMode := MC_HomingMode.MC_DefaultHoming; 
	fHomePosition		: LREAL := 0 	; // set position at homing
	fSafeVeloLimit		: LREAL	:= 360 	; // safe velocity limit [deg/sec]
	nEncTurnoverVal 	: LREAL := 360	; // encoder turnover value 
	tEnableDelay		: time 	:= T#0MS; // Time between axis enable command and motion command execution (0 := no delay active)	
	tDisabledelay		: TIME 	:= T#100MS; // Axis idle time before axis is disabled 
END_VAR
VAR 
	bActVeloReadValid 	: BOOL ; // velocity parameter read is valid 
	bActAccReadValid 	: BOOL ; // Acceleration parameter read is valid 
	bActDecReadValid 	: BOOL ; // Deceleration parameter read is valid 
	bActParamValid 		: BOOL ; // Parameter read is valid 
END_VAR
// Calculate device number
	ExecIdentifyDevice(nId,nParentId, E_ComponentTypes.Axis);

// ===== Message data set =====
	stFault.ComponentType		:= E_ComponentTypes.Axis ;
	
// ===== Write parameters =====
	stMParMaxAcc.nNumber		:= nLocationId + 1;
	stMParMaxAcc.sDiscription 	:= CONCAT(STR1 := sName, STR2:= ' hardware maximum accaleration (0 = HWMaximum)'); 
	stMParMaxAcc.sName			:= CONCAT(STR1 := sName, STR2:= 'Hard max aceleration');
	stMParMaxAcc.sType			:= 'MPar';
	stMParMaxAcc.sUnit			:= 'Units/Sec^2';
	
	stMParMaxDec.nNumber		:= nLocationId + 2;
	stMParMaxDec.sDiscription 	:= CONCAT(STR1 := sName, STR2:= ' hardware maximum deceleration(0 = HWMaximum)'); 
	stMParMaxDec.sName			:= CONCAT(STR1 := sName, STR2:= 'Hard max deceleration');
	stMParMaxDec.sType			:= 'MPar';
	stMParMaxDec.sUnit			:= 'Units/Sec^2';
	
	stMparMaxVelo.nNumber		:= nLocationId + 3;
	stMparMaxVelo.sDiscription 	:= CONCAT(STR1 := sName, STR2:= ' hardware maximum velocity'); 
	stMparMaxVelo.sName			:= CONCAT(STR1 := sName, STR2:= 'Hard max velocity');
	stMparMaxVelo.sType			:= 'MPar';
	stMparMaxVelo.sUnit			:= 'Units/Sec';

	refFbParHandler.CmdAddParameter(refParameter := stMParMaxAcc);
	refFbParHandler.CmdAddParameter(refParameter := stMParMaxDec);
	refFbParHandler.CmdAddParameter(refParameter := stMparMaxVelo);

// ===== set axis configuration =====	
	fMaxAcc	:= stMParMaxAcc.fValue;
	fMaxDec	:= stMParMaxDec.fValue;	
	fMaxVelo:= stMparMaxVelo.fValue;

	fCmdAcc 		:= fMaxAcc;
	fCmdDecc		:= fMaxDec;
// ===== Configure Axis =====
	// ***** Config Bits *****
		THIS^.bIcfCmdVelocityRpm	:= bIcfCmdVelocityRpm	; // Enable speed inputs in Rpm
		THIS^.bIcfEnableForward 	:= bIcfEnableForward 	; // Enable forward motion
		THIS^.bIcfEnablereverse		:= bIcfEnablereverse	; // Enable reverse motion
		THIS^.bIcfAlwaysEnable		:= bIcfAlwaysEnable		; // Always enable motor and brake if safety is ok
		THIS^.bIcfSimulationMode	:= bIcfSimulationMode 	; // Simulation mode is active [default set to False] 

	// ***** config homing Mode ***** 
 		THIS^.mcHomingMode 			:= mcHomingMode ; // set homing mode
 		THIS^.fHomePosition			:= fHomePosition;
	// ***** Velocity settings *****
		THIS^.fSafeVeloLimit 		:= fSafeVeloLimit ; // set maximum safe velocity	
	// ***** Time delay enable off *****
		THIS^.tEnableDelay		:= tEnableDelay	;
		THIS^.tDisableDelay 	:= tDisabledelay ;		

// ===== Set device type for manual control =====
	eDevType := E_Devices.Axis ;
		
// ===== reset axis state indicators ======
	bErrorActive 	:= FALSE;

// ====== Set init to done =======
	bInitOk	:= TRUE ;
END_METHOD

END_FUNCTION_BLOCK

// ---- Axis/FunctionBlocks/TwoVelocityControl/FB_DevTwoVelocityAxis.TcPOU
{attribute 'reflection'}
FUNCTION_BLOCK PUBLIC FB_DevTwoVelocityAxis EXTENDS FB_DevBase IMPLEMENTS iTwoDirectionalMotorWithFast
VAR // internal commands
	bCmdRunCW		: BOOL ; // run clockwise
	bCmdRunCWFast	: BOOL ; // Run fast
	bCmdRunCCW		: BOOL ; // run counter clockwise
	bCmdRunCCWFast	: BOOL ; // Run fast
	stManualControl	: st_ManualDigitalMotorControl ; // Manual control structure
END_VAR
VAR // Outputs
	qbRunCw			AT%Q* : BOOL ; // Output run clockwise
	qbRunCWFast		AT%Q* : BOOL ; // Output run clockwise Fast
	qbRunCCW 		AT%Q* : BOOL ; // Output run counter clockwise
	qbRunCCWFast	AT%Q* : BOOL ; // Output run Counter clockwise Fast	
END_VAR

SUPER^(refFbFault := refFbFault);

IF NOT bInitOk THEN
	RETURN;
END_IF

ExecSetOutputs();

METHOD PUBLIC CmdManual : BOOL
bCmdManual S= TRUE;

CmdManual := TRUE ;
END_METHOD

METHOD CmdRunCCW : BOOL
bCmdRunCCW := TRUE;

CmdRunCCW := qbRunCCW;
END_METHOD

METHOD CmdRunCCWFast : BOOL
bCmdRunCCWFast := TRUE;

CmdRunCCWFast := qbRunCCWFast;
END_METHOD

METHOD CmdRunCW : BOOL
bCmdRunCW := TRUE;

CmdRunCW := qbRunCW;
END_METHOD

METHOD CmdRunCWFast : BOOL
bCmdRunCWFast := TRUE;

CmdRunCWFast := qbRunCWFast;
END_METHOD

METHOD PUBLIC CmdSafeStop : BOOL
VAR_INPUT
END_VAR
CmdSafeStop := TRUE;

CmdSafeStop R= NOT qbRunCw;
CmdSafeStop R= NOT qbRunCWFast;
CmdSafeStop R= NOT qbRunCCW;
CmdSafeStop R= NOT qbRunCCWFast;	

qbRunCw			:= FALSE;
qbRunCWFast		:= FALSE;
qbRunCCW 		:= FALSE;
qbRunCCWFast	:= FALSE;
END_METHOD

METHOD INTERNAL ExecSetOutputs : BOOL
IF bSafetyOk THEN
	IF bManual THEN
		qbRunCw			:= stManualControl.bManRunCW;
		qbRunCWFast		:= stManualControl.bManRunCWFast;
		qbRunCCW 		:= stManualControl.bManRunCCw;
		qbRunCCWFast	:= stManualControl.bManRunCCWFast;
	ELSIF bEnable THEN
		qbRunCw			:= bCmdRunCW;
		qbRunCWFast		:= bCmdRunCWFast;
		qbRunCCW 		:= bCmdRunCCW;
		qbRunCCWFast	:= bCmdRunCCWFast;
	END_IF	
ELSE
	qbRunCw			:= FALSE;
	qbRunCWFast		:= FALSE;
	qbRunCCW 		:= FALSE;
	qbRunCCWFast	:= FALSE;	
END_IF

// reset all commands
bCmdRunCW		:= FALSE;
bCmdRunCWFast	:= FALSE;
bCmdRunCCW		:= FALSE;
bCmdRunCCWFast	:= FALSE;
stManualControl.bManRunCW 		:= FALSE;
stManualControl.bManRunCWFast 	:= FALSE;
stManualControl.bManRunCCw 		:= FALSE;
stManualControl.bManRunCCWFast	:= FALSE;

bCmdManual := FALSE;
END_METHOD

METHOD Init : BOOL
VAR_INPUT
	nId			: UDINT ; // Identification number of object
	nParentId	: UDINT ; // Id of higher level If aplicable (0 = no parent)
END_VAR
bInitOk := ExecIdentifyDevice(nId, nParentId, eComponentType := E_ComponentTypes.Axis);

// ===== Set device type for manual control =====
eDevType := E_Devices.TwoVelocityAxis ;

Init := bInitOk;
END_METHOD

END_FUNCTION_BLOCK

// ---- Buttons/Functions/FB_DevHMIButton.TcPOU
{attribute 'reflection'}
FUNCTION_BLOCK PUBLIC FB_DevHMIButton EXTENDS FB_DevBase // Button function for HMI 
VAR_INPUT
	Istatus			: BOOL	:= FALSE;// Digital sensor, Direct input status
	tDelay			: TIME 	:= T#5S	;// Time before delayed signal becomes active 
END_VAR
VAR_OUTPUT
	bFcoInputActive		: BOOL 			;// Digital sensor, Button active state
	bFcoDelay			: BOOL			;// Button, Delayed input status (3 seconds) 
	bFeStatus			: BOOL			;// Button, Falling edge of input signal	
	bReStatus			: BOOL			;// Button, Rising edge of input signal
	TetInputActive		: TIME			;// Button, Time elapsed while button is active
	bInvisible			: BOOL 			;// Button, Button is made invisible
	bDeactivate			: BOOL 			;// Button, Deactivate button 
END_VAR
VAR
	FB_delIStatus	: TON; // Timer function for delayed input status 
	FB_feIStatus	: F_TRIG; // generate falling edge pulse edge from Istatus
	FB_reIStatus	: R_TRIG; // generate falling edge pulse edge from Istatus
END_VAR

// Call base function
SUPER^(refFbFault := refFbFault);

// ***** Direct input when enabled *****
IF bEnable THEN 
	bFcoInputActive := Istatus ;
ELSE 
	bFcoInputActive := FALSE ;
END_IF

// ===== check if function is enabled =====
	IF NOT bEnable THEN 
		bInvisible 	:= TRUE ;
		bDeactivate	:= TRUE ;
		bFcoDelay	:= FALSE;
		RETURN;
	ELSE  
		bInvisible 	:= FALSE ;
		bDeactivate	:= FALSE ;
	END_IF

// ====== process functions if enabled ======
	// ***** Set Delayed inputs and time elapsed ****
		FB_delIStatus(	IN:= bFcoInputActive,
						PT:= tDelay , 
						Q=> bFcoDelay , 
						ET=> TetInputActive 
					  ); // Generate delayed input status from push button input status
	// ***** Edge triggers *****
		FB_feIStatus(CLK:= Istatus , Q=> bFeStatus ); // generate falling edge pulse on pushbutton input
		FB_reIStatus (Clk := Istatus , Q => bReStatus); // Generate rising edge from push button input signal

END_FUNCTION_BLOCK

// ---- Buttons/Functions/FB_DevPushButton.TcPOU
{attribute 'reflection'}
FUNCTION_BLOCK PUBLIC FB_DevPushButton EXTENDS Fb_DevDigitalInputFunctions
VAR_INPUT
END_VAR
VAR_OUTPUT
END_VAR
VAR
END_VAR

// set device type
IF eDevType = E_Devices.Undefined THEN 
	eDevType := E_Devices.DigitalSensor ;
END_IF

SUPER^(refFbFault := refFbFault);

END_FUNCTION_BLOCK

// ---- CounterCards/FunctionBlocks/KL1512/FB_DevKL1512.TcPOU
FUNCTION_BLOCK FB_DevKL1512 EXTENDS fb_devBase IMPLEMENTS iCounter
VAR
	nOldCount	   : UINT ; // Previous counter value 
	nBaseCount	   : UDINT; // Base counter
	ResetStep      : UINT;  // Current state of the reset sequence	
	bCmdResetValue : BOOL;  // The command to start the reset sequence
	bCmdResetDone  : BOOL;  // The reset has been processed
END_VAR
VAR // Inputs and outputs
	{info 'TODO: Add device state information and warnings (status is now unused var)'}
	{attribute 'analysis' := '-33'}
	State		AT%I* : USINT ; // status byte from card
	DataIn		AT%I* : UINT ;  // Data from the card 
	Ctrl 		AT%Q* : USINT ; // Control byte to card`
	DataOut 	AT%Q* : UINT ;  // Data to the card
END_VAR
VAR // Manual control
	stManualControl : st_ManualCounterControl;
END_VAR

ExecExtendCount();

ExecResetValue();

bCmdResetValue := FALSE;

METHOD PUBLIC CmdManual : BOOL
bCmdManual := TRUE;
stManualControl.nCount := nBaseCount + DataIn;;

IF stManualControl.bManSetValue THEN 
	// set counter to value
	DataOut	:= UDINT_TO_UINT(stManualControl.nManValue)	;
	Ctrl.5 	:= DataIn <> stManualControl.nManValue;
	
	stManualControl.bManSetValue R= DataIn = stManualControl.nManValue;
END_IF
END_METHOD

METHOD CmdReset : BOOL
VAR_INPUT
END_VAR
//Clear the control register
Ctrl := 0;

//Check the state is cleared
CmdReset := State = 0;
END_METHOD

METHOD CmdResetValue : BOOL
bCmdResetValue := TRUE;

CmdResetValue := bCmdResetDone;
END_METHOD

METHOD CmdSetValue : BOOL
VAR_INPUT
	Value	: UDINT;
END_VAR
nOldCount 	:= UDINT_TO_UINT(Value);
nBaseCount 	:= 0;

// set counter to value
DataOut	:= UDINT_TO_UINT(Value);
Ctrl.5 	:= DataIn <> Value;

CmdSetValue := DataIn = Value;
END_METHOD

PROPERTY CountValue : UDINT
GET
CountValue := nBaseCount + DataIn;
END_GET
END_PROPERTY

METHOD ExecExtendCount : BOOL
VAR_INPUT
END_VAR
IF nOldCount > DataIn AND NOT bCmdResetValue THEN
	nBaseCount := nbasecount + 16#10000 ;
END_IF
nOldCount := DataIn;
END_METHOD

METHOD ExecResetValue : BOOL
VAR_INPUT
END_VAR
CASE ResetStep OF
	0: (* Wait for the command to start *)
		IF (bCmdResetValue) THEN
			ResetStep := 10;
		END_IF
		
	10: (* Determine the next action *)
		IF (DataIn <> 0) THEN
			//Counter reset required
			ResetStep := 20;
		ELSE
			//Skip the reset procedure, just clear the internal counters
			ResetStep := 60;
		END_IF
		
	20: (* Set the clear bit *)
		Ctrl.1 := TRUE;
		ResetStep := 30;
		
	30: (* Wait untill the reset command has arrived *)
		IF (State.1) THEN
			ResetStep := 40;
		END_IF
		
	40: (* Release the clear bit *)
		Ctrl.1 := FALSE;
		ResetStep := 50;
		
	50: (* Validate the counter is cleared *)
		IF (DataIn = 0) THEN
			//Clear, proceed
			ResetStep := 60;
		ELSE
			//Not cleared, re-try
			ResetStep := 20;
		END_IF

	60: (* Clear the internal counters *)
		nOldCount := 0;
		nBaseCount := 0;
		ResetStep := 70;

	70: (* Indicate we are done *)
		bCmdResetDone := TRUE;
		IF (NOT bCmdResetValue) THEN
			bCmdResetDone := FALSE;
			ResetStep := 0;
		END_IF
END_CASE
END_METHOD

METHOD Init : BOOL
VAR_INPUT
END_VAR
//Clear the control register
Ctrl := 0;

//Wait untill the control register is cleared
bInitOk := State = 0;

Init := bInitOk;
END_METHOD

END_FUNCTION_BLOCK

// ---- CounterCards/FunctionBlocks/KL5151/FB_DevKL5151.TcPOU
{attribute 'reflection'}
FUNCTION_BLOCK FB_DevKL5151 EXTENDS FB_DevBase IMPLEMENTS iCounter
VAR_INPUT
	bInitAsCounterCard	: BOOL := FALSE; // (Default = FALSE) Use Terminal as encoder input (FALSE) or counter (TRUE) 
END_VAR
VAR CONSTANT // register values 
	WRITE_FEATURE_REGISTER 	: USINT := 16#E0; // write to register address command
	READ_FEATURE_REGISTER	: USINT := 16#A0; // Read feature register response  
END_VAR
VAR // Inputs and outputs
	Status		AT%I* : USINT ; // status byte from card
	Counter		AT%I* : UDINT ; // 
	Ctrl 		AT%Q* : USINT ; // Control byte to card`
	DataOut 	AT%Q* : UDINT ; // Set counter value
END_VAR
VAR // steppers
	InitStep : INT := 0; // init stepper
END_VAR
VAR // Manual control
	stManualControl : st_ManualCounterControl;
END_VAR

SUPER^(refFbFault := refFbFault);

METHOD PUBLIC CmdManual : BOOL
bCmdManual := TRUE;
stManualControl.nCount := Counter;

IF stManualControl.bManSetValue THEN 
	// set counter to value
	DataOut	:= stManualControl.nManValue	;
	Ctrl.2 	:= Counter <> stManualControl.nManValue;
	
	stManualControl.bManSetValue R= Counter = stManualControl.nManValue;
END_IF
END_METHOD

METHOD CmdReset : BOOL
VAR_INPUT
END_VAR
Ctrl.2 	:= FALSE;

CmdReset := NOT Status.2;
END_METHOD

METHOD CmdResetValue : BOOL // Reset the value of the counter card to 0
// set counter value to 0
DataOut	:= 0	;
Ctrl.2 	:= Counter <> 0;

CmdResetValue := Counter = 0;
END_METHOD

METHOD PUBLIC CmdSetValue : BOOL // Set the value of the counter card
VAR_INPUT
	Value	: UDINT;
END_VAR
// set counter to value
DataOut	:= Value	;
Ctrl.2 	:= Counter <> Value;

CmdSetValue := Counter = Value;
END_METHOD

PROPERTY PUBLIC CountValue : UDINT
GET
CountValue := Counter;
END_GET
END_PROPERTY

METHOD PUBLIC Init : BOOL
VAR_INPUT
	// Message location data
	nId				: UDINT ; // Identification number of object
	nParentId		: UDINT ; // Id of higher level If aplicable (0 = no parent)
END_VAR

IF bInitAsCounterCard THEN
//	{warning 'Counter function needs to be added to devices'}
	ExecIdentifyDevice(nId := nId, nParentId := nParentId, eComponentType := E_ComponentTypes.NA);
ELSE 
	ExecIdentifyDevice(nId := nId, nParentId := nParentId, eComponentType := E_ComponentTypes.Encoder);
END_IF

eDevType := E_Devices.KL5151;

// Check feature register against set function 
CASE InitStep OF 
	0: // check active feature register values
		Ctrl := READ_FEATURE_REGISTER;
		InitStep := initstep + 1;
	1: // Check if operation mode is correct If not set operation mode
		IF Status = READ_FEATURE_REGISTER THEN
			//Check if we are the requested mode
			IF Counter.15 = bInitAsCounterCard THEN 
				InitStep := 3;
			ELSE
				//Copy the current value into the output
				DataOut := Counter;
				//Set the encoder/counter bit as requested
				DataOut.15 := bInitAsCounterCard;
				//Give the command to write to the card
				Ctrl := WRITE_FEATURE_REGISTER;
				InitStep := 2;
			END_IF
		END_IF
	2: // Check if register was written	
		IF Status = READ_FEATURE_REGISTER THEN
			InitStep := 3;
		END_IF
		
	3: //Stop register access, return to normal
		//Copy the current value into the output
		Ctrl := Status;
		//Reset the register access bit
		Ctrl.7 := FALSE;
		InitStep := 4;
		
	4: //Check if the command was accepted
		IF Status.7 = 0 THEN
			InitStep := 10;
		END_IF
		
	10: // init done
		bInitOk := TRUE;
		
	ELSE
		;
END_CASE

Init := bInitOk;
END_METHOD

END_FUNCTION_BLOCK

// ---- Encoders/FunctionBlocks/FB_EncoderInput.TcPOU
{attribute 'reflection'}
FUNCTION_BLOCK FB_EncoderInput EXTENDS FB_EncoderBase
VAR_INPUT
END_VAR
VAR_OUTPUT
END_VAR
VAR
	iCounterValue 	AT%I*	: UDINT ;
	iDataError		AT%I*	: BOOL  ;	
	iFrameError		AT%I*	: BOOL  ;
	iPowerFailure	AT%I*	: BOOL  ; 
	iSyncError		AT%I*	: BOOL  ;
	
	nScaledValue		: LREAL ; // Only scaled value for internal use
	nValueWithOffset	: LREAL ; // scaled value with added offset
	fOldPos				: LREAL ; // Old position
	
END_VAR

// ====== Check device status ======
	CheckBoxStatus();

// ====== Scale Output value ======
	nScaledValue := UDINT_TO_LREAL(iCounterValue) / fPulsesPerUnit ;

// ====== Invert ======
	IF bIcfInverted THEN 
		nScaledValue := nScaledValue * -1;
	END_IF
	
// ====== Add offset ======= 
	nValueWithOffset := nScaledValue + fOffset ;
	
// ====== Caclulate velocity =====
	IF Sys_Variables.Pulse100ms THEN 
		nVelocity 	:= (nOutPosition - fOldPos) * 10 ;
		fOldPos		:= nOutPosition;
	END_IF
	
// ====== Set Outputs =======
	nOutPosition 	:= nValueWithOffset ;
	nOutRaw			:= iCounterValue	;

METHOD PRIVATE CheckBoxStatus : BOOL
VAR_INPUT
END_VAR
IF iDataError THEN 
	stFault.Active 			:= TRUE ;
	stFault.Discription		:= CONCAT(sName, ' Encoder Data error');
	stFault.MessageNumber	:= E_MessageNumbers.FF_ComunicationFault;
	stFault.FaultType		:= E_FaultTypes.FF;
ELSIF iFrameError THEN 
	stFault.Active 			:= TRUE ;
	stFault.Discription		:= CONCAT(sName, ' Encoder frame error');
	stFault.MessageNumber	:= E_MessageNumbers.FF_ComunicationFault;
	stFault.FaultType		:= E_FaultTypes.FF;
ELSIF iPowerFailure THEN 
	stFault.Active 			:= TRUE ;
	stFault.Discription		:= CONCAT(sName, ' Encoder Power failure');
	stFault.MessageNumber	:= E_MessageNumbers.FF_ComunicationFault;
	stFault.FaultType		:= E_FaultTypes.FF;
ELSIF iSyncError THEN 
	stFault.Active 			:= TRUE ;
	stFault.Discription		:= CONCAT(sName, ' Encoder synchronisation error');
	stFault.MessageNumber	:= E_MessageNumbers.FF_ComunicationFault;
	stFault.FaultType		:= E_FaultTypes.FF;
END_IF
END_METHOD

METHOD PUBLIC FastTask : BOOL
VAR_INPUT
END_VAR
END_METHOD

END_FUNCTION_BLOCK

// ---- HardwareDiagnostics/FB_ELModuleDiag.TcPOU
{attribute 'reflection'}
FUNCTION_BLOCK PUBLIC FB_ELModuleDiag
VAR_INPUT
END_VAR
VAR_OUTPUT
	bError 	:	BOOL ; // Module is in error
	sErrorDiscription : STRING ; // module error discription 
END_VAR
VAR
END_VAR

END_FUNCTION_BLOCK

// ---- Sensors/AnalogInput/FunctionBlocks/FB_DevAnalogInputScaled.TcPOU
{attribute 'reflection'}
FUNCTION_BLOCK PUBLIC FB_DevAnalogInputScaled EXTENDS FB_DevAnalogInput
VAR_INPUT
END_VAR
VAR_OUTPUT
END_VAR
VAR
	fGainFactor 	: LREAL	:= 1	;
	nOfset			: INT	:= 0	;
END_VAR

SUPER^(refFbFault := refFbFault);

METHOD ExecSetFeedback : BOOL
VAR
	nCalibValue	: INT ; 
END_VAR
// Offset 
IF bCmdSimulate THEN 
	nCalibValue := fSimValue + nOfset ;
ELSE
	nCalibValue := inHwInput + nOfset ;
END_IF

fValue := INT_TO_LREAL(nCalibValue) / fGainFactor;

ExecSetFeedback := TRUE;
END_METHOD

METHOD PUBLIC SetScaling : BOOL 
VAR_INPUT
	fMaxValue	: LREAL ; 	// Maximum input value after scaling, e.g. 100%, 0 = no scaling (gain = hardware limit / fMaxValue)  
	fOfset		: LREAL ;	// offset value (fvalue = (gain * hwvalue) + fOfset)
END_VAR
// calculate gain 
IF fMaxValue =0 THEN 
	fGainFactor := 1 ;
ELSE 
	fGainFactor := nLimitMax / fMaxValue ;
END_IF

nOfset := LREAL_TO_INT(fOfset * fGainFactor) ;

SetScaling := TRUE;
END_METHOD

END_FUNCTION_BLOCK

// ---- Sensors/AnalogInput/FunctionBlocks/FB_DevHDAnalogInAutoCalibrate.TcPOU
{attribute 'reflection'}
FUNCTION_BLOCK PUBLIC FB_DevHDAnalogInAutoCalibrate EXTENDS FB_DevHDAnalogInputScaled
VAR_INPUT
END_VAR
VAR_OUTPUT
END_VAR
VAR
END_VAR

SUPER^(refFbFault := refFbFault);

METHOD PUBLIC CmdCalibrateNull : BOOL
VAR_INPUT
END_VAR
// set offset to calibrate to null
nOfset := - inHwInput ;

CmdCalibrateNull := TRUE;
END_METHOD

METHOD PUBLIC CmdCalilbrateValue : BOOL // calibrate gain factor to actual value (warning calibrate to null before calibrating to value)
VAR_INPUT
	fCalibrationValue	: LREAL ; // Active input value to sensor (calibration setpoint)
END_VAR
// set gain from current value
fGainFactor := DINT_TO_LREAL(inHwInput + nOfset) / fCalibrationValue ; 

CmdCalilbrateValue := TRUE;
END_METHOD

END_FUNCTION_BLOCK

// ---- Sensors/AnalogInput/FunctionBlocks/FB_DevHDAnalogInputScaled.TcPOU
{attribute 'reflection'}
FUNCTION_BLOCK PUBLIC FB_DevHDAnalogInputScaled EXTENDS FB_DevHDAnalogInput
VAR_INPUT
END_VAR
VAR_OUTPUT
END_VAR
VAR
	fGainFactor 	: LREAL	:= 1	;
	nOfset			: DINT	:= 0	;
END_VAR

SUPER^(refFbFault := refFbFault);

METHOD ExecSetFeedback : BOOL
VAR
	nCalibValue	: DINT ; 
END_VAR
// Offset 
IF bCmdSimulate THEN 
	nCalibValue := fSimValue + nOfset ;
ELSE
	nCalibValue := inHwInput + nOfset ;
END_IF

fValue := DINT_TO_LREAL(nCalibValue) / fGainFactor;
END_METHOD

METHOD PUBLIC SetScaling : BOOL 
VAR_INPUT
	fMaxValue	: LREAL ; 	// Maximum input value after scaling, e.g. 100%, 0 = no scaling (gain = hardware limit / fMaxValue)  
	fOfset		: LREAL ;	// offset value (fvalue = (gain * hwvalue) + fOfset)
END_VAR
// calculate gain 
IF fMaxValue =0 THEN 
	fGainFactor := 1 ;
ELSE 
	fGainFactor := nLimitMax / fMaxValue ;
END_IF

nOfset := LREAL_TO_DINT(fOfset * fGainFactor) ;

SetScaling := TRUE ;
END_METHOD

END_FUNCTION_BLOCK

// ---- Sensors/AnalogInput/FunctionBlocks/FB_DevHDAnalogInput.TcPOU
{attribute 'reflection'}
FUNCTION_BLOCK PUBLIC FB_DevHDAnalogInput EXTENDS FB_DevBase
VAR_INPUT
	bCmdSimulate	: BOOL 	:= FALSE ;// Simulate sensor Input 
	fSimValue		: DINT	:= 0 ;// Simulated sensor state
END_VAR
VAR_OUTPUT
	fValue	: LREAL := 0 ; // Analog input value (LREAL)
END_VAR
VAR
	nLimitMin			: DINT := Utilities_Library.GVL_FixedValues.nDINTMINVALUE	; // Initial value is set to integer minimum value for use with normal def analog inputs 
	nLimitMax 			: DINT := Utilities_Library.GVL_FixedValues.nDINTMAXVALUE 	; // Initial value is set to integer minimum value for use with high def analog inputs
	inHwInput 	AT%I* 	: DINT ; // Hardware connection
	inStatus	AT%I* 	: BYTE; // input card hardware status
END_VAR

// Set device type
eDevType := E_Devices.AnalogSensor ;

// Call base function
SUPER^(refFbFault := refFbFault);

// Check Hardware connection
CheckHardware();

// set feedback
ExecSetFeedback();

METHOD CheckHardware : BOOL
VAR_INPUT
END_VAR
// Check for hardware faults
IF inStatus.0 THEN // signal under range
	stFault.Active			:= TRUE 							;
	stFault.MessageNumber	:= E_MessageNumbers.CF_FeedbackFault 	;
	stFault.Discription		:= CONCAT( sName, 'Signal under Range' )	;
	stFault.FaultType		:= E_FaultTypes.CF 					;
	bErrorActive			:= TRUE 							;
END_IF

IF inStatus.1 THEN // signal over range
	stFault.Active			:= TRUE 							;
	stFault.MessageNumber	:= E_MessageNumbers.CF_FeedbackFault 	;
	stFault.Discription		:= CONCAT( sName, 'Signal over Range' )	;
	stFault.FaultType		:= E_FaultTypes.CF 					;
	bErrorActive			:= TRUE 							;
END_IF

IF inStatus.6 THEN // general Error bit
	stFault.Active			:= TRUE 							;
	stFault.MessageNumber	:= E_MessageNumbers.FF_Unknown 	;
	stFault.Discription		:= CONCAT( sName, 'Hardware General Error' )	;
	stFault.FaultType		:= E_FaultTypes.FF 					;
	bErrorActive			:= TRUE 							;
END_IF
END_METHOD

METHOD ExecSetFeedback : BOOL
VAR_INPUT
END_VAR
IF bCmdSimulate THEN 
	fValue := fSimValue ;
ELSE
	fValue := DINT_TO_LREAL(inHwInput);
END_IF

ExecSetFeedback := TRUE;
END_METHOD

METHOD PUBLIC Init : BOOL
VAR_INPUT
	// Location data for messages  
	nId			: UDINT ; // Identification number of object
	nParentId	: UDINT ; // Id of higher level If aplicable (0 = no parent)
END_VAR
// ====== Set init to true =====
	bInitOk	:= TRUE ; 

// ====== Calculate device id =====
	bInitOk :=	ExecIdentifyDevice(nId,nParentId, E_ComponentTypes.AnInput) AND bInitOk;

// ====== Set feedback =====
	Init := bInitOk ;
END_METHOD

END_FUNCTION_BLOCK

// ---- Sensors/AnalogInput/FunctionBlocks/FB_DevAnalogInAutoCalibrate.TcPOU
{attribute 'reflection'}
FUNCTION_BLOCK PUBLIC FB_DevAnalogInAutoCalibrate EXTENDS FB_DevAnalogInputScaled
VAR_INPUT
END_VAR
VAR_OUTPUT
END_VAR
VAR
END_VAR

SUPER^(refFbFault := refFbFault);

METHOD PUBLIC CmdCalibrateNull : BOOL
VAR_INPUT
END_VAR
// set offset to calibrate to null
nOfset := - inHwInput ;
END_METHOD

METHOD PUBLIC CmdCalilbrateValue : BOOL // calibrate gain factor to actual value (warning calibrate to null before calibrating to value)
VAR_INPUT
	fCalibrationValue	: LREAL ; // Active input value to sensor (calibration setpoint)
END_VAR
// set gain from current value
fGainFactor := INT_TO_LREAL(inHwInput + nOfset) / fCalibrationValue ;
END_METHOD

END_FUNCTION_BLOCK

// ---- Sensors/FootPedals/FunctionBlocks/FB_EfkaEB301A_FootPedal.TcPOU
{attribute 'reflection'}
FUNCTION_BLOCK PUBLIC FB_EfkaEB301A_FootPedal EXTENDS FB_DevBase
VAR_OUTPUT
	ePedalInputStep		: E_FootpedalPos	:= 0 ;
	bRTrigtoReverse1 	: BOOL := FALSE ; // rising edge trigger when pedal moves from 0 to -1 or Idle to reverse 1 
	bRTrigtoReverse2 	: BOOL := FALSE ; // rising edge trigger when pedal moves from 1 to -2 or reverse 1 to reverse 2 
	bRTrigtoForward1 	: BOOL := FALSE ; // rising edge trigger when pedal moves from 0 to 1 or idle to forward 1 
	bRTrigtoForward2 	: BOOL := FALSE ; // rising edge trigger when pedal moves from 0 to 1 or forward to forward 2 
END_VAR
VAR
	// ===== greycode switches from footpedal =====
	I_GreyCodeA AT%I* : BOOL	; // Greycode input a from foot pedal 
	I_GreyCodeB AT%I* : BOOL	; // Greycode input a from foot pedal 
	I_GreyCodeC AT%I* : BOOL	; // Greycode input a from foot pedal 
	I_GreyCodeD AT%I* : BOOL	; // Greycode input a from foot pedal 
	nGreyCodetotal	: BYTE ; // all greycode switches combined
	// ==== decimal value =====
	ePreviousPedalInput	: E_FootpedalPos	:= 0 ;
END_VAR

// ===== Read input from pedal =====
ACT_ConvertGreycode();

// ===== Create edge flanks for functions =====
ACT_CreateEdges();

ACTION ACT_ConvertGreycode:
// ===== Combine greycode sensors =====
nGreyCodetotal.0 := I_GreyCodeA ;
nGreyCodetotal.1 := I_GreyCodeB ;
nGreyCodetotal.2 := I_GreyCodeC ;
nGreyCodetotal.3 := I_GreyCodeD ;

// ==== Convert greycode decimal to speed steps =====
// this only makes sense in EFKA world but anyway let's convert it to our own sense

CASE nGreyCodetotal OF 								  // DCBA
	03: ePedalInputStep := E_FootpedalPos.eReverse2	; // 0011
	01: ePedalInputStep := E_FootpedalPos.eReverse1	; // 0001
	00: ePedalInputStep := E_FootpedalPos.eIdle		; // 0000
	02: ePedalInputStep := E_FootpedalPos.eForward0	; // 0010
	06: ePedalInputStep := E_FootpedalPos.eForward1	; // 0110
 	07: ePedalInputStep := E_FootpedalPos.eForward2	; // 0111
	05: ePedalInputStep := E_FootpedalPos.eForward3	; // 0101
	04: ePedalInputStep := E_FootpedalPos.eForward4	; // 0100
	12:	ePedalInputStep := E_FootpedalPos.eForward5	; // 1100
	13:	ePedalInputStep := E_FootpedalPos.eForward6	; // 1101
	15: ePedalInputStep := E_FootpedalPos.eForward7	; // 1111
	14: ePedalInputStep := E_FootpedalPos.eForward8	; // 1110
	10: ePedalInputStep := E_FootpedalPos.eForward9	; // 1010
	11: ePedalInputStep := E_FootpedalPos.eForward10; // 1011
	09: ePedalInputStep := E_FootpedalPos.eForward11; // 1001
	08: ePedalInputStep := E_FootpedalPos.eForward12; // 1000
	ELSE
		ePedalInputStep := E_FootpedalPos.eFalse 	;
END_CASE
END_ACTION

ACTION ACT_CreateEdges:
// ===== create edges on which functions can be triggerd =====
CASE ePedalInputStep OF
	E_FootpedalPos.eReverse2:
		bRTrigtoReverse2 := ePreviousPedalInput = E_FootpedalPos.eReverse1 ;
	E_FootpedalPos.eReverse1:
		bRTrigtoReverse1 := ePreviousPedalInput = E_FootpedalPos.eIdle ;
	E_FootpedalPos.eForward0:
		bRTrigtoForward1 := ePreviousPedalInput = E_FootpedalPos.eIdle ;
	E_FootpedalPos.eForward1: 
		bRTrigtoForward2 := ePreviousPedalInput = E_FootpedalPos.eForward0 ; 
END_CASE 

// write previous pedal input 
ePreviousPedalInput := ePedalInputStep ;
END_ACTION

METHOD PUBLIC Init : BOOL
VAR_INPUT
	// Location data for messages  
	nId			: UDINT ; // Identification number of object
	nParentId	: UDINT ; // Id of higher level If aplicable (0 = no parent)
END_VAR
// ====== Set init to true =====
	bInitOk	:= TRUE ; 

// ====== Calculate device id =====
	bInitOk :=	ExecIdentifyDevice(nId,nParentId, E_ComponentTypes.NA) AND bInitOk;

// ====== Set feedback =====
	Init := bInitOk;
END_METHOD

END_FUNCTION_BLOCK
